// TIA Portal V16 export
// export: Created 2021-11-12T13:32:40.1658868Z, ExportSetting WithDefaults, DisplayName Totally Integrated Automation Portal, DisplayVersion V16 Update 3, DisplayName TIA Portal Version Control Interface, DisplayVersion V16 Update 2, DisplayName TIA Portal Openness, DisplayVersion V16 Update 3, DisplayName SINAMICS Startdrive Advanced, DisplayVersion V16 Update 5, DisplayName SINAMICS Startdrive G130, G150, S120, S150, SINAMICS MV, S210, DisplayVersion V16 Update 5, DisplayName SINAMICS Startdrive G110M, G120, G120C, G120D, G120P, G115D, DisplayVersion V16 Update 5, DisplayName STEP 7 Professional, DisplayVersion V16 Update 3, DisplayName STEP 7 Safety, DisplayVersion V16, DisplayName WinCC UA Professional, DisplayVersion V16 Update 3
DATA_BLOCK "HMI_PARAM_2R2"   // DB2114
{ S7_Optimized_Access := 'TRUE' }
VERSION : 0.1
// stored: AutoNumber false, DBAccessibleFromOPCUA true, IsOnlyStoredInLoadMemory false, IsRetainMemResEnabled false, IsWriteProtectedInAS false, MemoryReserve 100
   VAR
      xxxxx___BinarySensors___xxxxx : Byte;
      "CM01-BL01_4" : "UDT_CH_DI_Parameter";   // Proplachovací nádrž 2 Vysoká hladina Varování
      "CM01-BL01_5" : "UDT_CH_DI_Parameter";   // Proplachovací nádrž 2 Vysoká hladina Max
      xxxxx___BinaryOthers___xxxxx : Byte;
      PwrOK : "UDT_CH_DI_Parameter";
      "000UH11-SF13" : "UDT_CH_DI_Parameter";   // Okamžitý stop Robot 2R2
      "000UH11-SF10" : "UDT_CH_DI_Parameter";   // Robot 2R2 Proplach
      "000UH11-SF11" : "UDT_CH_DI_Parameter";   // Robot 2R2 Nástřik
      xxxxx___AnalogueSensors___xxxxx : Byte;
      xxxxx___Drives___xxxxx : Byte;
      RO01 : "UDT_RobotABB_Parameter";   // Robot
      RC01 : "UDT_DriveRobotABB_Parameter";   // Controller
      Lubricating : "UDT_DriveRobotABB_Parameter";   // Lubricating
      xxxxx___Others___xxxxx : Byte;
      xxxxx___Alarms___xxxxx : Byte;
      RO01_Timeout : "UDT_DI_Mon_Parameter";   // Robot job active for too long
      RO01_LubStartErr : "UDT_DI_Mon_Parameter";   // Lubrication job did not start (robot did not move)
      "CM01-BL01_4_alarm" : "UDT_DI_Mon_Parameter";   // Proplachovací nádrž 1 Vysoká hladina Varování
      "CM01-BL01_5_alarm" : "UDT_DI_Mon_Parameter";   // Proplachovací nádrž 1 Vysoká hladina Max
      xxxxx___SftyAlarms___xxxxx : Byte;
      ES { S7_SetPoint := 'True'} : "UDT_DI_Mon_Parameter";   // E-stop
   END_VAR
BEGIN
END_DATA_BLOCK
